// TIA Portal V19 export
FUNCTION_BLOCK "Block_1"   // FB2, FBD
{ S7_Optimized_Access := 'TRUE' }
// stored: MemoryReserve 100, SetENOAutomatically false
   VAR_INPUT
      V1 : Bool;
      v2 : Bool;
   END_VAR
   VAR
      Program_Alarm_1 { S7_SetPoint := 'True'} : Program_Alarm;
   END_VAR
BEGIN

REGION Network 1
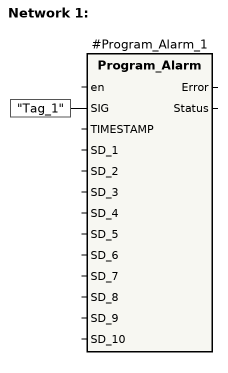
   #Program_Alarm_1(SIG := "Tag_1");   // Program_Alarm
END_REGION
END_FUNCTION_BLOCK
